{attribute 'GeneratedUsingTerminal: EP3632-0001-0016'}
{attribute addProperty BoxType "EP3632-0001-0016"}
{attribute addProperty Id "UnderrangeBOOL1OverrangeBOOL1Limit_1BYTE1Limit_2BYTE1ErrorBOOL1Sync_errorBOOL1TxPDO_StateBOOL1TxPDO_ToggleBOOL1"}
{attribute addProperty CRC "2960470870"}
{attribute addProperty Size "8"}
TYPE STATUS_B0753356 :
STRUCT
	{attribute addProperty Name "Underrange"}
	Underrange : BOOL;
	{attribute addProperty Name "Overrange"}
	Overrange : BOOL;
	{attribute addProperty Name "Limit_1"}
	Limit_1 : BYTE;
	{attribute addProperty Name "Limit_2"}
	Limit_2 : BYTE;
	{attribute addProperty Name "Error"}
	Error : BOOL;
	{attribute addProperty Name "Sync_error"}
	Sync_error : BOOL;
	{attribute addProperty Name "TxPDO_State"}
	TxPDO_State : BOOL;
	{attribute addProperty Name "TxPDO_Toggle"}
	TxPDO_Toggle : BOOL;
END_STRUCT
END_TYPE

(* stored: Version 1.2.0.0, ProductVersion 3.1.4024.9
   DUT STATUS_B0753356: Id {08e92170-716d-4dfa-9ca3-e2f8403b3e88} *)
